// LS Electric XG5000 project: 동남87
// PLC NewPLC
// module base 0 slot 0: 입출력 모듈:XBC-DN/DP14E (DC 24V 입력 8점, 트랜지스터 출력 6점)

PROGRAM NewProgram (task: 스캔 프로그램)

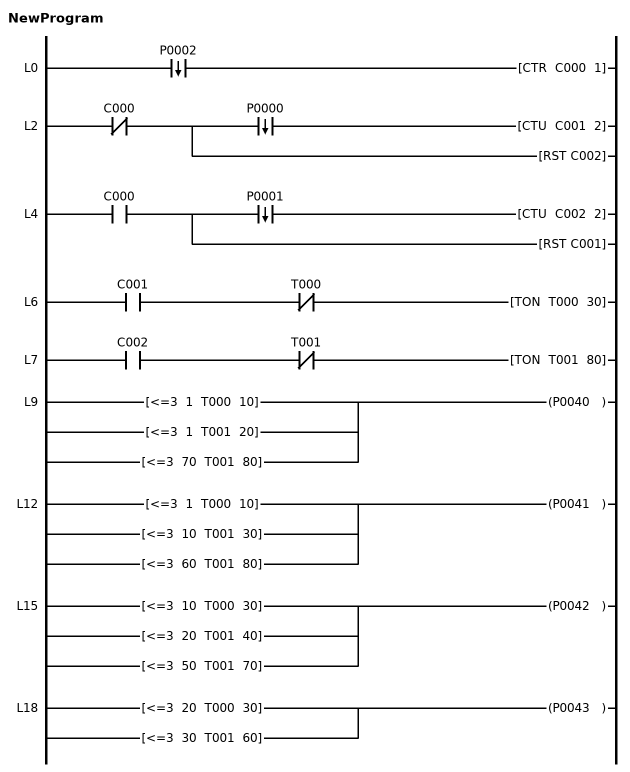
; L0
LOADN     P0002
CTR       C000 1
; L2
LOAD NOT  C000
MPUSH
ANDN      P0000
CTU       C001 2
MPOP
RST       C002
; L4
LOAD      C000
MPUSH
ANDN      P0001
CTU       C002 2
MPOP
RST       C001
; L6
LOAD      C001
AND NOT   T000
TON       T000 30
; L7
LOAD      C002
AND NOT   T001
TON       T001 80
; L9
LOAD<=3   1 T000 10
OR<=3     1 T001 20
OR<=3     70 T001 80
OUT       P0040
; L12
LOAD<=3   1 T000 10
OR<=3     10 T001 30
OR<=3     60 T001 80
OUT       P0041
; L15
LOAD<=3   10 T000 30
OR<=3     20 T001 40
OR<=3     50 T001 70
OUT       P0042
; L18
LOAD<=3   20 T000 30
OR<=3     30 T001 60
OUT       P0043